// TIA Portal V19 export
TYPE "SpeedMachine_CIn_Manager"
// stored: Access Published
   STRUCT
      EnableStopDoorOpeningReq : Bool := TRUE;
      EnableStopInPhase : Bool := TRUE;
      EnableStopProgrammed : Bool := TRUE;
      Control_ON : Bool := FALSE;
      Bwd : Bool := FALSE;
      Fwd : Bool := FALSE;
      Vel : LReal := 100.0;
      Acc : LReal := 100.0;
      Dec : LReal := 100.0;
   END_STRUCT;
END_TYPE
